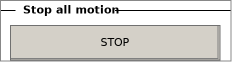
VISUALIZATION VISU_BaseAxis_Stop  // 232x62
VAR_IN_OUT
	axis : BaseAxis;
    axisWidget : BaseAxisWidget;
END_VAR
    Button (10,25 210x35), "STOP", input disabled if: axis.processes.stop.statuses.enabledStatus.disabled
        OnMouseClick: execute { axis.processes.stop.do_request := TRUE; }
    Label (20,0 95x20), "Stop all motion"
    Line (115,10) (230,10)
    Line (0,10) (15,10)
END_VISUALIZATION

(* stored: Version 1.1.0.1, ProductVersion 3.1.4019.2
   Visu VISU_BaseAxis_Stop: Id {990e13b8-bf5a-4283-b079-f6476b962f04} *)
